TYPE ST_AnalogInput :
STRUCT
	stStatus 	AT %I* : ST_AnalogInputStatus;
	nValue		AT %I* : INT;	
END_STRUCT
END_TYPE

(* stored: Version 1.1.0.1, ProductVersion 3.1.4024.10
   DUT ST_AnalogInput: Id {a0ce17ac-e8d5-4661-804c-b62193a832da} *)
